// TIA Portal V16 export
// export: Created 2025-12-30T17:36:37.644539Z, ExportSetting WithDefaults, DisplayName Totally Integrated Automation Portal, DisplayVersion V16, DisplayName TIA Portal Version Control Interface, DisplayVersion V16, DisplayName TIA Portal Openness, DisplayVersion V16, DisplayName STEP 7 Professional, DisplayVersion V16, DisplayName STEP 7 Safety, DisplayVersion V16, DisplayName WinCC Professional, DisplayVersion V16
ORGANIZATION_BLOCK "Main"   // OB1, LAD, ProgramCycle
TITLE = "Main Program Sweep (Cycle)"
{ S7_Optimized_Access := 'TRUE' }
VERSION : 0.1
// stored: AutoNumber true, IsIECCheckEnabled false, SetENOAutomatically false
   VAR_INPUT
      Initial_Call : Bool;   // Initial call of this OB
      Remanence : Bool;   // =True, if remanent data are available
   END_VAR
   VAR_TEMP
      temp : Real;
   END_VAR
BEGIN

REGION Network 1
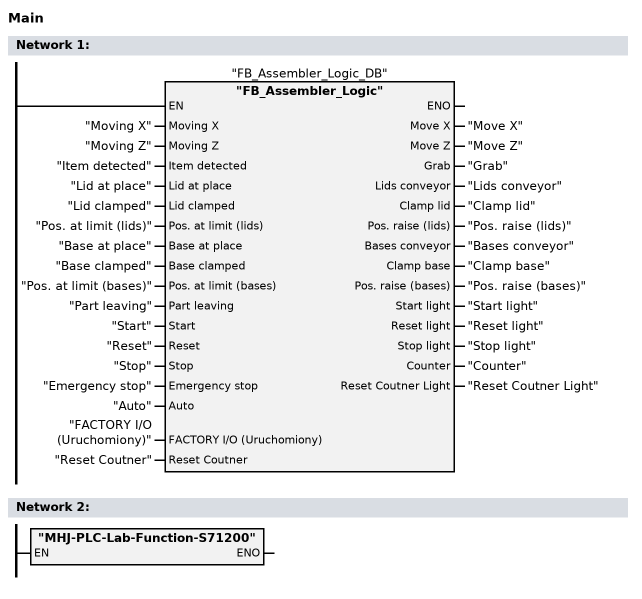
   RUNG wire#powerrail
      "FB_Assembler_Logic_DB"("Moving X" := "Moving X", "Moving Z" := "Moving Z", "Item detected" := "Item detected", "Lid at place" := "Lid at place", "Lid clamped" := "Lid clamped", "Pos. at limit (lids)" := "Pos. at limit (lids)", "Base at place" := "Base at place", "Base clamped" := "Base clamped", "Pos. at limit (bases)" := "Pos. at limit (bases)", "Part leaving" := "Part leaving", Start := "Start", Reset := "Reset", Stop := "Stop", "Emergency stop" := "Emergency stop", Auto := "Auto", "FACTORY I/O (Uruchomiony)" := "FACTORY I/O (Uruchomiony)", "Reset Coutner" := "Reset Coutner", "Move X" => "Move X", "Move Z" => "Move Z", Grab => "Grab", "Lids conveyor" => "Lids conveyor", "Clamp lid" => "Clamp lid", "Pos. raise (lids)" => "Pos. raise (lids)", "Bases conveyor" => "Bases conveyor", "Clamp base" => "Clamp base", "Pos. raise (bases)" => "Pos. raise (bases)", "Start light" => "Start light", "Reset light" => "Reset light", "Stop light" => "Stop light", "Counter" => "Counter", "Reset Coutner Light" => "Reset Coutner Light")
   END_RUNG
   // the same network as SCL:
   "FB_Assembler_Logic_DB"("Moving X" := "Moving X",   // "FB_Assembler_Logic"
                           "Moving Z" := "Moving Z",
                           "Item detected" := "Item detected",
                           "Lid at place" := "Lid at place",
                           "Lid clamped" := "Lid clamped",
                           "Pos. at limit (lids)" := "Pos. at limit (lids)",
                           "Base at place" := "Base at place",
                           "Base clamped" := "Base clamped",
                           "Pos. at limit (bases)" := "Pos. at limit (bases)",
                           "Part leaving" := "Part leaving",
                           Start := "Start",
                           Reset := "Reset",
                           Stop := "Stop",
                           "Emergency stop" := "Emergency stop",
                           Auto := "Auto",
                           "FACTORY I/O (Uruchomiony)" := "FACTORY I/O (Uruchomiony)",
                           "Reset Coutner" := "Reset Coutner",
                           "Move X" => "Move X",
                           "Move Z" => "Move Z",
                           Grab => "Grab",
                           "Lids conveyor" => "Lids conveyor",
                           "Clamp lid" => "Clamp lid",
                           "Pos. raise (lids)" => "Pos. raise (lids)",
                           "Bases conveyor" => "Bases conveyor",
                           "Clamp base" => "Clamp base",
                           "Pos. raise (bases)" => "Pos. raise (bases)",
                           "Start light" => "Start light",
                           "Reset light" => "Reset light",
                           "Stop light" => "Stop light",
                           "Counter" => "Counter",
                           "Reset Coutner Light" => "Reset Coutner Light");
END_REGION

REGION Network 2
   RUNG wire#powerrail
      "MHJ-PLC-Lab-Function-S71200"()
   END_RUNG
   // the same network as SCL:
   "MHJ-PLC-Lab-Function-S71200"();
END_REGION
END_ORGANIZATION_BLOCK
